TYPE ST_MachineOutputs :
STRUCT
    bSafetyRunRequest                  : BOOL;
    bSafetyResetRequest                : BOOL;
    bSafetyErrorAcknowledgementRequest : BOOL;
    bAirSupplyEnable                   : BOOL;
    bMainDoorLockRequest               : BOOL;
    bIndexRotatePortA                  : BOOL;
    bIndexStopPortB                    : BOOL;
    bIndexSupportExtend                : BOOL;
    bIndexSupportRetract               : BOOL;

    bStation1SupportExtend             : BOOL;
    bStation1SupportRetract            : BOOL;
    bStation2SupportExtend             : BOOL;
    bStation2SupportRetract            : BOOL;
    bStation3SupportExtend             : BOOL;
    bStation3SupportRetract            : BOOL;
	// Patch Dispensing
	bPatchDispenserAir 					: BOOL;
	bPatchVerticalDown 					: BOOL;
	bPatchVerticalUp   					: BOOL;


    // Vision Station / Flipping tooling
    bVisionHorizontalBack              : BOOL;
    bVisionHorizontalFront             : BOOL;
    bVisionVerticalUp                  : BOOL;
    bVisionVerticalDown                : BOOL;
    bVisionLimitOff                    : BOOL;
    bVisionLimitOn                     : BOOL;
    bVisionGripClose                   : BOOL;
    bVisionGripOpen                    : BOOL;
    bVisionRotate0                     : BOOL;
    bVisionRotate180                   : BOOL;

    bHeatStakeHeadLock                 : BOOL;
    bHeatStakeHeadUnlock               : BOOL;
    bHeatStakeHeadDown                 : BOOL;
    bHeatStakeHeadUp                   : BOOL;
    iHeatStakePressureRaw              : INT;
    bLedStart                          : BOOL;
    bLedReset                          : BOOL;
    bLedPass                           : BOOL;
    bLedFail                           : BOOL;
    bInternalLight                     : BOOL;
    bNestLight                         : BOOL;
    uiHeatStakePwm1Raw                 : UINT;
    uiHeatStakePwm2Raw                 : UINT;
	
	//camera
	sBatchNumber			: STRING;
	sDate					: STRING;
	bPatchOk				: BOOL;
	bClickPart				: ARRAY [1..2] OF BOOL;
	bBluePartOk				: BOOL;
	bPBUBPartOk				: BOOL;
	bGeneralPass			: BOOL;
	bGeneralFail			: BOOL;
	bProgramLoadComplete	: BOOL;
	bResultsReady			: BOOL;
	bRunStatus				: BOOL;
	
END_STRUCT
END_TYPE

(* stored: Version 1.1.0.1, ProductVersion 3.1.4026.18
   DUT ST_MachineOutputs: Id {54b65e3e-4603-4fb6-b710-aae3df30541a} *)
